FUNCTION_BLOCK Model (* Composite Function Block Type *)
  (* Standard: 61499-2 *)
  (* Version 0.0, 5/29/2016, Andrei, nxtControl GmbH, template *)
  PACKAGE Main;
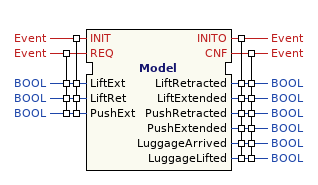
  EVENT_INPUT
    INIT WITH LiftExt, LiftRet, PushExt; (* Initialization Request *)
    REQ WITH LiftExt, LiftRet, PushExt; (* Normal Execution Request *)
  END_EVENT
  EVENT_OUTPUT
    INITO WITH LiftRetracted, LiftExtended, PushRetracted, PushExtended, LuggageArrived, LuggageLifted; (* Initialization Confirm *)
    CNF WITH LiftRetracted, LiftExtended, PushRetracted, PushExtended, LuggageArrived, LuggageLifted; (* Execution Confirmation *)
  END_EVENT
  VAR_INPUT
    LiftExt : BOOL;
    LiftRet : BOOL;
    PushExt : BOOL;
  END_VAR
  VAR_OUTPUT
    LiftRetracted : BOOL;
    LiftExtended : BOOL; (* Output event qualifier *)
    PushRetracted : BOOL;
    PushExtended : BOOL;
    LuggageArrived : BOOL;
    LuggageLifted : BOOL;
  END_VAR
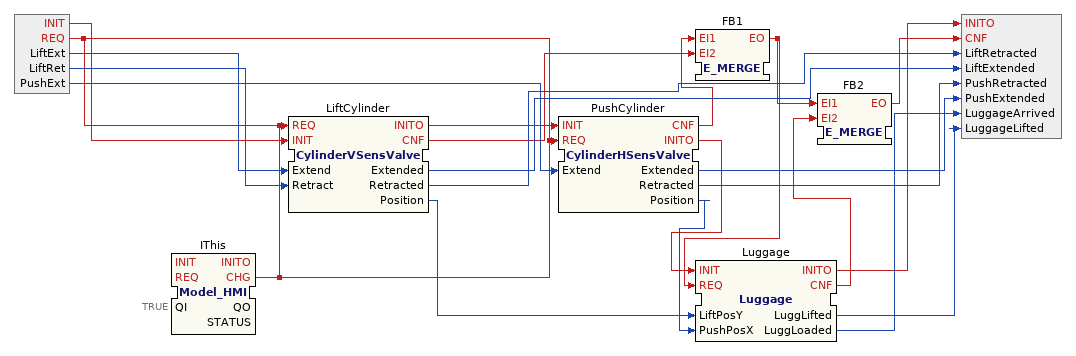
  FBS
    LiftCylinder : CylinderVSensValve;
    PushCylinder : CylinderHSensValve;
    IThis : Model_HMI(QI := TRUE);
    Luggage : Luggage;
    FB1 : E_MERGE;
    FB2 : E_MERGE;
  END_FBS
  EVENT_CONNECTIONS
    REQ TO LiftCylinder.REQ;
    INIT TO LiftCylinder.INIT;
    LiftCylinder.INITO TO PushCylinder.INIT;
    IThis.CHG TO LiftCylinder.REQ;
    IThis.CHG TO PushCylinder.REQ;
    PushCylinder.CNF TO FB1.EI1;
    LiftCylinder.CNF TO FB1.EI2;
    PushCylinder.INITO TO Luggage.INIT;
    Luggage.INITO TO INITO;
    REQ TO PushCylinder.REQ;
    FB2.EO TO CNF;
    FB1.EO TO Luggage.REQ;
    FB1.EO TO FB2.EI1;
    Luggage.CNF TO FB2.EI2;
  END_CONNECTIONS
  DATA_CONNECTIONS
    LiftCylinder.Extended TO LiftExtended;
    LiftCylinder.Retracted TO LiftRetracted;
    PushCylinder.Extended TO PushExtended;
    PushCylinder.Retracted TO PushRetracted;
    LiftCylinder.Position TO Luggage.LiftPosY;
    PushCylinder.Position TO Luggage.PushPosX;
    Luggage.LuggLifted TO LuggageLifted;
    Luggage.LuggLoaded TO LuggageArrived;
    LiftExt TO LiftCylinder.Extend;
    LiftRet TO LiftCylinder.Retract;
    PushExt TO PushCylinder.Extend;
  END_CONNECTIONS
END_FUNCTION_BLOCK
